// TIA Portal project "CTRL_HSC_fonksiyonu" (V18)

(* hardware
DEVICE "S7-1200 station_1"  S7-1200 Station
   slot 0: "Rack_0"  S7-1200 Rack  Rack  V1.0
   slot 1: "PLC_1"  CPU 1214C DC/DC/DC  6ES7 214-1AG40-0XB0  V4.6
*)

// ===== PLC "PLC_1"  CPU 1214C DC/DC/DC =====

VAR_GLOBAL   // PLC tag table "Default tag table"
   "Tag_1" AT %I0.4 : Bool;
   "Tag_2" AT %M20.0 : Bool;
   "Tag_3" AT %MW50 : Word;
   "HSC5 DEĞERİ" AT %ID1016 : DWord;
   "HSC5 ATAMA" AT %MD30 : DWord;
   "Tag_4" AT %I0.0 : Bool;
   "Tag_5" AT %Q0.0 : Bool;
   "Tag_6" AT %Q0.1 : Bool;
   "Tag_7" AT %I0.1 : Bool;
   "Tag_8" AT %Q0.3 : Bool;
   "Tag_9" AT %Q1.0 : Bool;
   "Tag_10" AT %Q1.1 : Bool;
END_VAR

ORGANIZATION_BLOCK "Main"   // OB1, LAD, ProgramCycle
TITLE = "Main Program Sweep (Cycle)"
{ S7_Optimized_Access := 'TRUE' }
VERSION : 0.1
   VAR_INPUT
      Initial_Call : Bool;   // Initial call of this OB
      Remanence : Bool;   // =True, if remanent data are available
   END_VAR
BEGIN

REGION Network 1
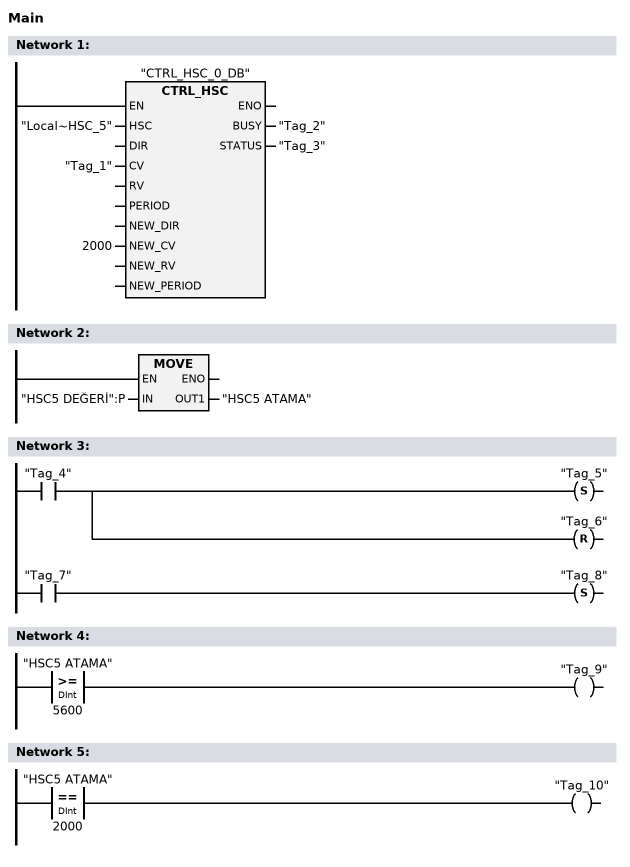
   "CTRL_HSC_0_DB"(HSC := "Local~HSC_5", CV := "Tag_1", NEW_CV := 2000, BUSY => "Tag_2", STATUS => "Tag_3");   // CTRL_HSC
END_REGION

REGION Network 2
   RUNG wire#powerrail
      Move(in := "HSC5 DEĞERİ":P, out1 => "HSC5 ATAMA")
   END_RUNG
   // the same network as SCL:
   "HSC5 ATAMA" := "HSC5 DEĞERİ":P;
END_REGION

REGION Network 3
   RUNG wire#powerrail
      Contact( "Tag_4" )
      wire#w1
      S_Coil( "Tag_5" )
   END_RUNG
   RUNG wire#w1
      R_Coil( "Tag_6" )
   END_RUNG
   RUNG wire#powerrail
      Contact( "Tag_7" )
      S_Coil( "Tag_8" )
   END_RUNG
   // the same network as SCL:
   IF "Tag_4" THEN
       "Tag_5" := TRUE;
       "Tag_6" := FALSE;
   END_IF;
   IF "Tag_7" THEN "Tag_8" := TRUE; END_IF;
END_REGION

REGION Network 4
   RUNG wire#powerrail
      { S7_Templates := "SrcType := DInt" } GE_Contact(in1 := "HSC5 ATAMA", in2 := 5600)
      Coil( "Tag_9" )
   END_RUNG
   // the same network as SCL:
   "Tag_9" := "HSC5 ATAMA" >= 5600;
END_REGION

REGION Network 5
   RUNG wire#powerrail
      { S7_Templates := "SrcType := DInt" } EQ_Contact(in1 := "HSC5 ATAMA", in2 := 2000)
      Coil( "Tag_10" )
   END_RUNG
   // the same network as SCL:
   "Tag_10" := "HSC5 ATAMA" = 2000;
END_REGION
END_ORGANIZATION_BLOCK